(* IEC 61131-3 sources: matiec/tests/hang, 7 files *)

(* ---- end_transition_in_function.st ---- *)
FUNCTION F : INT
VAR_INPUT a : INT; END_VAR
  F := a;
END_TRANSITION
END_FUNCTION

(* ---- action_bad_name.st ---- *)
PROGRAM P
VAR a : BOOL; END_VAR
INITIAL_STEP S0: END_STEP
TRANSITION FROM S0 TO S0 := a; END_TRANSITION
ACTION 1: a := x.y; END_ACTION
END_PROGRAM

(* ---- resource_junk.st ---- *)
PROGRAM P
VAR a : BOOL; END_VAR
a := TRUE;
END_PROGRAM
CONFIGURATION C
RESOURCE R ON PLC
  TASK T(INTERVAL := T#10ms, PRIORITY := 0);
  PROGRAM I WITH T : P;
END_RESOURCE
END_IF
END_CONFIGURATION

(* ---- sfc_network_junk.st ---- *)
PROGRAM P
VAR a : BOOL; END_VAR
INITIAL_STEP S0: END_STEP
TRANSITION FROM S0 TO S0 := a; END_TRANSITION
END_IF
END_PROGRAM

(* ---- sfc_network_junk2.st ---- *)
PROGRAM P
VAR a : BOOL; END_VAR
INITIAL_STEP S0: END_STEP .
END_PROGRAM

(* ---- transition_bad_destination.st ---- *)
PROGRAM P
VAR a : BOOL; END_VAR
INITIAL_STEP S0: END_STEP
TRANSITION FROM S0 TO 1 := x.y; END_TRANSITION
END_PROGRAM

(* ---- transition_hang.st ---- *)
PROGRAM P
VAR a : BOOL; END_VAR
INITIAL_STEP S0: END_STEP
TRANSITION FROM S0 TO S0 := x.y; END_TRANSITION
END_PROGRAM
